% RSLogix 500 project Automated O2 Sensor Calibration System using PLC.RSS, saved by version 8.30.00.16 %
PROJECT "UNTITLED"    % processor: Bul.1763 MicroLogix 1100 Series B %

PROGRAM FILES
  LAD 2   6 rungs
  LAD 3 "IO"  5 rungs
  LAD 4 "VALV_CTRL"  3 rungs
  LAD 5 "TIMERS"  8 rungs
  LAD 8 "SCAL ALRM"  2 rungs

DATA FILES
  O0 OUTPUT  4 elements
  I1 INPUT  6 elements
  S2 STATUS  66 elements
  B3 BINARY  2 elements
  T4 TIMER  4 elements
  C5 COUNTER  2 elements
  R6 CONTROL  1 elements
  N7 INTEGER  12 elements
  F8 FLOAT  9 elements

LADDER 2
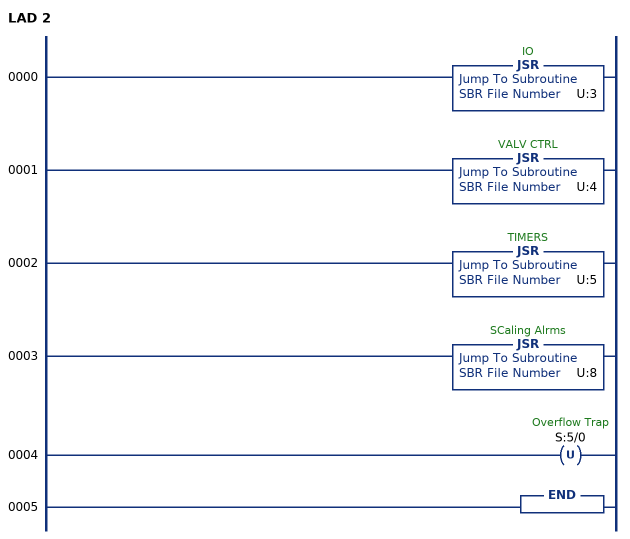
% Rung: 0 %
SOR JSR U:3 EOR
%   U:3  "IO" %
% Rung: 1 %
SOR JSR U:4 EOR
%   U:4  "VALV CTRL" %
% Rung: 2 %
SOR JSR U:5 EOR
%   U:5  "TIMERS" %
% Rung: 3 %
SOR JSR U:8 EOR
%   U:8  "SCaling Alrms" %
% Rung: 4 %
SOR OTU S:5/0 EOR
%   S:5/0  "Overflow Trap" %
% Rung: 5 %
SOR END EOR

LADDER 3 "IO"
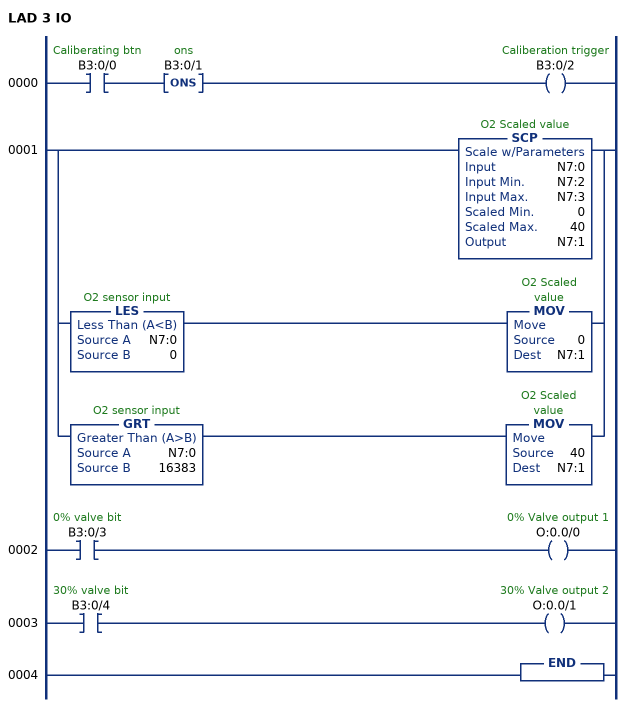
% Rung: 0 %
SOR XIC B3:0/0 ONS B3:0/1 OTE B3:0/2 EOR
%   B3:0/0  "Caliberating btn" %
%   B3:0/1  "ons" %
%   B3:0/2  "Caliberation trigger" %
% Rung: 1 %
SOR BST SCP N7:0 N7:2 N7:3 0 40 N7:1 NXB LES N7:0 0 MOV 0 N7:1 NXB GRT N7:0 16383 MOV 40 N7:1 BND EOR
%   N7:0  "O2 sensor input" %
%   N7:2  "o2 ip MIn" %
%   N7:3  "O2 IP Max" %
%   N7:1  "O2 Scaled value" %
% Rung: 2 %
SOR XIC B3:0/3 OTE O:0.0/0 EOR
%   B3:0/3  "0% valve bit" %
%   O:0.0/0  "0% Valve output 1" %
% Rung: 3 %
SOR XIC B3:0/4 OTE O:0.0/1 EOR
%   B3:0/4  "30% valve bit" %
%   O:0.0/1  "30% Valve output 2" %
% Rung: 4 %
SOR END EOR

LADDER 4 "VALV_CTRL"
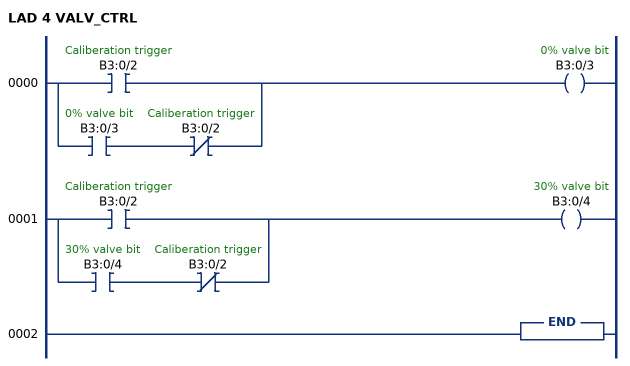
% Rung: 0 %
SOR BST XIC B3:0/2 NXB XIC B3:0/3 XIO B3:0/2 BND OTE B3:0/3 EOR
%   B3:0/2  "Caliberation trigger" %
%   B3:0/3  "0% valve bit" %
% Rung: 1 %
SOR BST XIC B3:0/2 NXB XIC B3:0/4 XIO B3:0/2 BND OTE B3:0/4 EOR
%   B3:0/2  "Caliberation trigger" %
%   B3:0/4  "30% valve bit" %
% Rung: 2 %
SOR END EOR

LADDER 5 "TIMERS"
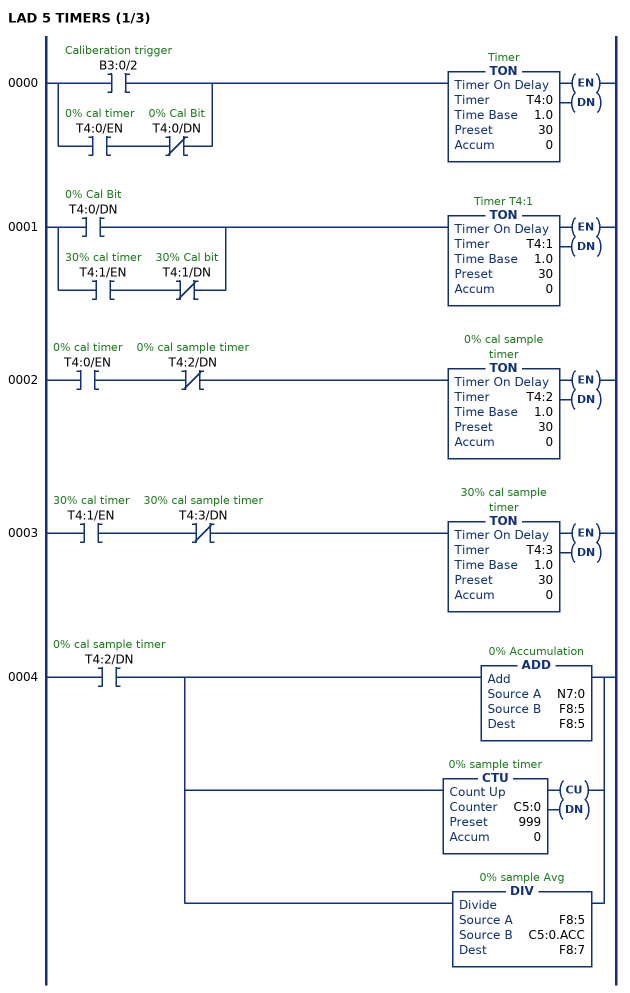
% Rung: 0 %
SOR BST XIC B3:0/2 NXB XIC T4:0/EN XIO T4:0/DN BND TON T4:0 1.0 30 0 EOR
%   B3:0/2  "Caliberation trigger" %
%   T4:0/EN  "0% cal timer" %
%   T4:0/DN  "0% Cal Bit" %
%   T4:0  "Timer" %
% Rung: 1 %
SOR BST XIC T4:0/DN NXB XIC T4:1/EN XIO T4:1/DN BND TON T4:1 1.0 30 0 EOR
%   T4:0/DN  "0% Cal Bit" %
%   T4:1/EN  "30% cal timer" %
%   T4:1/DN  "30% Cal bit" %
%   T4:1  "Timer T4:1" %
% Rung: 2 %
SOR XIC T4:0/EN XIO T4:2/DN TON T4:2 1.0 30 0 EOR
%   T4:0/EN  "0% cal timer" %
%   T4:2  "0% cal sample timer" %
% Rung: 3 %
SOR XIC T4:1/EN XIO T4:3/DN TON T4:3 1.0 30 0 EOR
%   T4:1/EN  "30% cal timer" %
%   T4:3/DN  "30% cal sample timer" %
%   T4:3  "30% cal sample timer" %
% Rung: 4 %
SOR XIC T4:2/DN BST ADD N7:0 F8:5 F8:5 NXB CTU C5:0 999 0 NXB DIV F8:5 C5:0.ACC F8:7 BND EOR
%   T4:2  "0% cal sample timer" %
%   N7:0  "O2 sensor input" %
%   F8:5  "0% Accumulation" %
%   C5:0  "0% sample timer" %
%   F8:7  "0% sample Avg" %

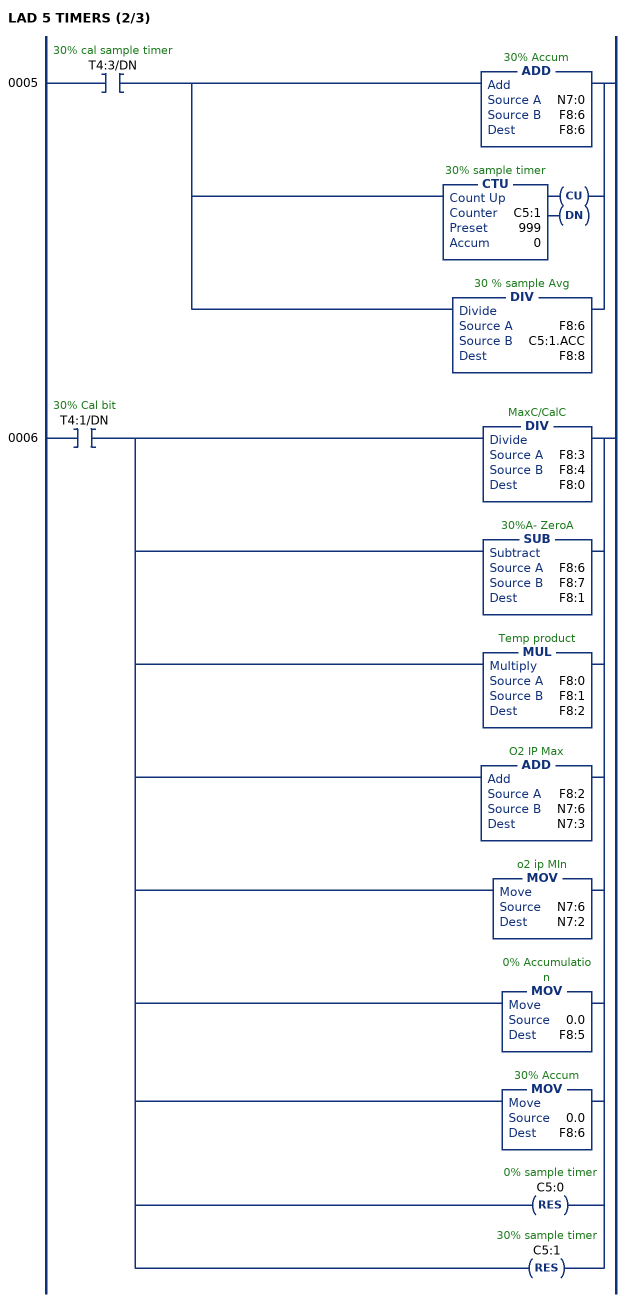
% Rung: 5 %
SOR XIC T4:3/DN BST ADD N7:0 F8:6 F8:6 NXB CTU C5:1 999 0 NXB DIV F8:6 C5:1.ACC F8:8 BND EOR
%   T4:3/DN  "30% cal sample timer" %
%   N7:0  "O2 sensor input" %
%   F8:6  "30% Accum" %
%   C5:1  "30% sample timer" %
%   C5:1.ACC  "30% sample AVg" %
%   F8:8  "30 % sample Avg" %
% Rung: 6 %
SOR XIC T4:1/DN BST DIV F8:3 F8:4 F8:0 NXB SUB F8:6 F8:7 F8:1 NXB MUL F8:0 F8:1 F8:2 NXB ADD F8:2 N7:6 N7:3 NXB MOV N7:6 N7:2 NXB MOV 0.0 F8:5 NXB MOV 0.0 F8:6 NXB RES C5:0 NXB RES C5:1 BND EOR
%   T4:1/DN  "30% Cal bit" %
%   F8:3  "MaxC/CalC" %
%   F8:0  "MaxC/CalC" %
%   F8:6  "30% Accum" %
%   F8:7  "0% sample Avg" %
%   F8:1  "30%A- ZeroA" %
%   F8:2  "Temp product" %
%   N7:6  "o2 ip MIn" %
%   N7:3  "O2 IP Max" %
%   N7:2  "o2 ip MIn" %
%   F8:5  "0% Accumulation" %
%   C5:0  "0% sample timer" %
%   C5:1  "30% sample timer" %

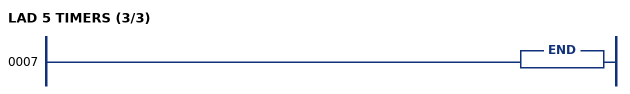
% Rung: 7 %
SOR END EOR

LADDER 8 "SCAL ALRM"
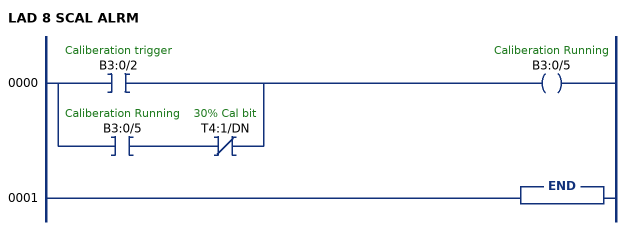
% Rung: 0 %
SOR BST XIC B3:0/2 NXB XIC B3:0/5 XIO T4:1/DN BND OTE B3:0/5 EOR
%   B3:0/2  "Caliberation trigger" %
%   B3:0/5  "Caliberation Running" %
%   T4:1/DN  "30% Cal bit" %
% Rung: 1 %
SOR END EOR

OTHER DOCUMENTED ADDRESSES
  B3:0/6  "Control bit 1"
  B3:0/7  "Contro bit 2"
  B3:1/0  "ONS"
  B3:1/1  "Cal Active"
  B3:1/2  "Stage 1 Active"
  B3:1/3  "Stage 2 Active"
  B3:1/4  "ONS"
  B3:1/5  "ONS"
  B3:2/0  B3  "0% Valve close"
  B3:2/1  "30% Valve Open"
  I:0.0/0  "O2 sensor input"
  I:0.0/1  "Calliberation push button"
  I:1.0/0  "Valve0_Feedback"
  I:1.0/1  "Valve1_Feedback"
  N7:10  "ACCUMULATE 0% SAMPLES"
  N7:11  "ACCUMULATE 30% SAMPLES"
  O:0.0  "0% gas valve"
  O:0.0/2  "Control output 1"
  O:0.0/3  "Valve output 1"
  O:0.1  "30% gas valve"
  U:6  "SAM logic"
  U:7  "CALC LOGIC"

DATA TABLE (non-zero values as saved)
DATA T4
% .PRE .ACC %
% T4:0 % 30 0
% T4:1 % 30 0
% T4:2 % 30 0
% T4:3 % 30 0
DATA C5
% .PRE .ACC %
% C5:0 % 999 0
% C5:1 % 999 0
DATA N7
% N7:0 % 0 0 0 16383 0 0 0 0 0 0
DATA F8
% F8:0 % 0 0 0 40 30
